// TwinCAT 3 PLC project ACSenLib
// Title: ACSenLib
// Company: EBC
// ProjectVersion: 0.1
// ProgramVersion: 3.1.4026.18
// project tree:
//   DUTs/ S_InputVar.TcDUT
//   Interfaces/ I_HumiditySensor.TcIO, I_TemperatureSensor.TcIO, I_VolumeFlowSensor.TcIO
//   Sensors/ FB_ElectrMeas_EL3413.TcPOU, FB_HumiditySensor_EL3054.TcPOU, FB_Optiflux5000_EL3022.TcPOU, FB_PT100_EL3202.TcPOU, FB_PT100_EL3214.TcPOU, FB_TroxDrall_EL3062.TcPOU, FB_VolumeFlow_EL3054.TcPOU, FB_Vortex_EL3112.TcPOU

// ---- DUTs/S_InputVar.TcDUT
TYPE S_InputVar :
STRUCT
	(*	
RealVar=IntVarInput*RealParaM+RealParaC

RealParaMinWert>=RealVar>=RealParaMaxWert

IntVarOutput=(RealVar-RealParaC)/RealParaM

*)	

	IntVarInput AT %I*	:INT ; //Input von Klemme (z.B. 2100)
	RealVar 			:REAL; //Wert als REAL/Float/Single (z.B. 21.00)
	
	RealParaM 			:REAL; //Parameter M
	RealParaC 			:REAL; //Parameter C
	
	RealParaMaxVal 	:REAL; //Maximaler Wert des nativen Wertes (z.B. 10V, 20mA)
	RealParaMinVal 	:REAL; //Minimaler Wert des nativen Wertes (z.B. 0V, 4mA)	
	
END_STRUCT
END_TYPE

// ---- Interfaces/I_HumiditySensor.TcIO
INTERFACE I_HumiditySensor

PROPERTY Humidity : REAL
GET
END_GET
END_PROPERTY

END_INTERFACE

// ---- Interfaces/I_TemperatureSensor.TcIO
INTERFACE I_TemperatureSensor

PROPERTY Temperature : REAL
GET
END_GET
END_PROPERTY

END_INTERFACE

// ---- Interfaces/I_VolumeFlowSensor.TcIO
INTERFACE I_VolumeFlowSensor

PROPERTY VolumeFlow : REAL
GET
END_GET
END_PROPERTY

END_INTERFACE

// ---- Sensors/FB_ElectrMeas_EL3413.TcPOU
FUNCTION_BLOCK FB_ElectrMeas_EL3413
VAR
	fCurInt_P1 AT %I* : DINT;
	fCurInt_P2 AT %I* : DINT;
	fCurInt_P3 AT %I* : DINT;
	fCur_P1 : REAL;
	fCur_P2 : REAL;
	fCur_P3 : REAL;
	fmCur : REAL := 0.000004; //Multiplier Current
	fVolInt_P1 AT %I* : DINT;
	fVolInt_P2 AT %I* : DINT;
	fVolInt_P3 AT %I* : DINT;
	fVol_P1 : REAL;
	fVol_P2 : REAL;
	fVol_P3 : REAL;
	fmVol : REAL := 0.0001; //Multiplier voltage
	fPowerInt_P1 AT %I* : DINT;
	fPowerInt_P2 AT %I* : DINT;
	fPowerInt_P3 AT %I* : DINT;
	fPower_P1 : REAL;
	fPower_P2: REAL;
	fPower_P3 : REAL;
	fmPow : REAL := 0.04; //Multiplier power 
	fPower_total :REAL;
END_VAR

// Electrical measurements with EL3413

PROPERTY Power_P1 : REAL
GET
Power_P1 := THIS^.fPower_P1;
END_GET
END_PROPERTY

PROPERTY Power_P2 : REAL
GET
Power_P2 := THIS^.fPower_P2;
END_GET
END_PROPERTY

PROPERTY Power_P3 : REAL
GET
Power_P3 := THIS^.fPower_P3;
END_GET
END_PROPERTY

PROPERTY Power_total : REAL
GET
Power_total := THIS^.fPower_total;
END_GET
END_PROPERTY

METHOD Read
VAR_INPUT
END_VAR
//Read Current
fCur_P1 := DINT_TO_REAL(fCurInt_P1) * fmCur; 
fCur_P2 := DINT_TO_REAL(fCurInt_P2) * fmCur; 
fCur_P3 := DINT_TO_REAL(fCurInt_P3) * fmCur;

//Voltage
fVol_P1 := DINT_TO_REAL(fVolInt_P1) * fmVol;
fVol_P2 := DINT_TO_REAL(fVolInt_P2) * fmVol;
fVol_P3 := DINT_TO_REAL(fVolInt_P3) * fmVol;

//Power
fPower_P1 := DINT_TO_REAL(fPowerInt_P1) * fmPow;
fPower_P2 := DINT_TO_REAL(fPowerInt_P2) * fmPow;
fPower_P3 := DINT_TO_REAL(fPowerInt_P3) * fmPow;

fPower_total := fPower_P1 + fPower_P2 + fPower_P3;
END_METHOD

END_FUNCTION_BLOCK

// ---- Sensors/FB_HumiditySensor_EL3054.TcPOU
FUNCTION_BLOCK FB_HumiditySensor_EL3054 IMPLEMENTS I_HumiditySensor
VAR_INPUT
END_VAR
VAR_OUTPUT
END_VAR
VAR
	//Property Real value
	fHumidity : REAL;
	//Raw value
	HumRaw AT %I* : INT;
	//Convertion parameters
	m : REAL := 0.00305185071; //Multiplier for convertion
END_VAR

// Humidity measurement with rotronic HygroFlex 5 
// https://www.rotronic.com/de/catalog/product/view/id/299/s/hygroflex5-hf5-hlk-messumformer/category/12/

PROPERTY Humidity : REAL
GET
fHumidity := m* INT_TO_REAL(HumRaw);
Humidity := THIS^.fHumidity;
END_GET
END_PROPERTY

END_FUNCTION_BLOCK

// ---- Sensors/FB_Optiflux5000_EL3022.TcPOU
FUNCTION_BLOCK FB_Optiflux5000_EL3022 IMPLEMENTS I_VolumeFlowSensor
VAR_INPUT
END_VAR
VAR_OUTPUT
END_VAR
VAR								
	//Property Real value
	fVolFlow : REAL;
	//Raw value
	VolFlowRaw AT %I* : INT;
	//Convertion parameters
	m : REAL := 0.1098666341; //Multiplier for convertion
END_VAR

// Volume Flow measurement with Krohne Optiflux 5000
// https://www.krohne.com/de-de/produkte/durchflussmesstechnik/komponenten-und-zusaetzliche-betriebsmittel-fuer-die-durchflussmessung/messwertaufnehmer/optiflux-5000

PROPERTY VolumeFlow : REAL
GET
fVolFlow := m * INT_TO_REAL(VolFlowRaw);
VolumeFlow := THIS^.fVolFlow;
END_GET
END_PROPERTY

END_FUNCTION_BLOCK

// ---- Sensors/FB_PT100_EL3202.TcPOU
FUNCTION_BLOCK FB_PT100_10DIN_EL3202 IMPLEMENTS I_TemperatureSensor
VAR
	//Property Real value
	fTemperature : REAL;
	//Raw value
	TempRaw AT %I* : INT;
	//Convertion parameters
	m : REAL := 0.01; //Multiplier for convertion
END_VAR

//Temperature measurement: PT 100 1/10 DIN + EL3202:(0010,0020,0030) 4-wire

PROPERTY Temperature : REAL
GET
fTemperature := INT_TO_REAL(TempRaw) * m;
Temperature := THIS^.fTemperature;
END_GET
END_PROPERTY

END_FUNCTION_BLOCK

// ---- Sensors/FB_PT100_EL3214.TcPOU
FUNCTION_BLOCK FB_PT100_EL3214 IMPLEMENTS I_TemperatureSensor
VAR_INPUT
END_VAR
VAR_OUTPUT
END_VAR
VAR
	//Property Real value
	fTemperature : REAL;
	//Raw value
	TempRaw AT %I* : INT;
	//Convertion parameters
	m : REAL := 0.1; //Multiplier for convertion
END_VAR

//Temperature measurement: PT 100 1/10 DIN + EL3214: 3-wire

PROPERTY Temperature : REAL
GET
fTemperature := INT_TO_REAL(TempRaw) * m;
Temperature := THIS^.fTemperature;
END_GET
END_PROPERTY

END_FUNCTION_BLOCK

// ---- Sensors/FB_TroxDrall_EL3062.TcPOU
FUNCTION_BLOCK FB_TroxDrall_EL3062 IMPLEMENTS I_VolumeFlowSensor
VAR_INPUT
END_VAR
VAR_OUTPUT
END_VAR
VAR
	//Propertie Real value
	fVolumeFlow : REAL;
	//Raw value
	VolumeFlowRaw AT %I* : INT;
	//Convertion parameters
	m : REAL := 0.0444959849; //Multiplier for convertion
END_VAR

// Air Volume Flow measurement with Trox Drallauslass

PROPERTY VolumeFlow : REAL
GET
//Read volume flow
fVolumeFlow := m * INT_TO_REAL (VolumeFlowRaw); 
VolumeFlow := This^.fVolumeFlow;
END_GET
END_PROPERTY

END_FUNCTION_BLOCK

// ---- Sensors/FB_VolumeFlow_EL3054.TcPOU
FUNCTION_BLOCK FB_VolumeFlow_EL3054 IMPLEMENTS I_VolumeFlowSensor
VAR_INPUT
END_VAR
VAR_OUTPUT
END_VAR
VAR
	//Property Real value
	fVolFlow : REAL;
	//Raw value
	VolFlowRaw AT %I* : INT;
	//Convertion parameters
	m : REAL := 0.000366222026; //Multiplier for convertion
END_VAR

PROPERTY VolumeFlow : REAL
GET
fVolFlow := m * INT_TO_REAL(VolFlowRaw);
VolumeFlow := THIS^.fVolFlow;
END_GET
END_PROPERTY

END_FUNCTION_BLOCK

// ---- Sensors/FB_Vortex_EL3112.TcPOU
FUNCTION_BLOCK FB_Vortex_EL3112 IMPLEMENTS I_VolumeFlowSensor
VAR_INPUT
END_VAR
VAR_OUTPUT
END_VAR
VAR								
	//Property Real value
	fVolFlow : REAL;
	//Raw value
	VolFlowRaw AT %I* : INT;
	//Convertion parameters
	m : REAL := 0.00305185071; //Multiplier for convertion
END_VAR

// Volume Flow measurement with Grundfos Vortex sensor

PROPERTY VolumeFlow : REAL
GET
fVolFlow := m * INT_TO_REAL(VolFlowRaw);
VolumeFlow := THIS^.fVolFlow;
END_GET
END_PROPERTY

END_FUNCTION_BLOCK
